# EPICS autosave request: xx_auto_scalcout_settings.req
$(P)$(S).A
$(P)$(S).B
$(P)$(S).C
$(P)$(S).D
$(P)$(S).E
$(P)$(S).F
$(P)$(S).G
$(P)$(S).H
$(P)$(S).I
$(P)$(S).J
$(P)$(S).K
$(P)$(S).L
$(P)$(S).INPA
$(P)$(S).INPB
$(P)$(S).INPC
$(P)$(S).INPD
$(P)$(S).INPE
$(P)$(S).INPF
$(P)$(S).INPG
$(P)$(S).INPH
$(P)$(S).INPI
$(P)$(S).INPJ
$(P)$(S).INPK
$(P)$(S).INPL
$(P)$(S).AA
$(P)$(S).BB
$(P)$(S).CC
$(P)$(S).DD
$(P)$(S).EE
$(P)$(S).FF
$(P)$(S).GG
$(P)$(S).HH
$(P)$(S).II
$(P)$(S).JJ
$(P)$(S).KK
$(P)$(S).LL
$(P)$(S).INAA
$(P)$(S).INBB
$(P)$(S).INCC
$(P)$(S).INDD
$(P)$(S).INEE
$(P)$(S).INFF
$(P)$(S).INGG
$(P)$(S).INHH
$(P)$(S).INII
$(P)$(S).INJJ
$(P)$(S).INKK
$(P)$(S).INLL
$(P)$(S).CALC
$(P)$(S).OCAL
$(P)$(S).SCAN
$(P)$(S).PREC
$(P)$(S).ODLY
$(P)$(S).OEVT
$(P)$(S).OOPT
$(P)$(S).DOPT
$(P)$(S).IVOA
$(P)$(S).IVOV
$(P)$(S).OUT
$(P)$(S).FLNK
$(P)$(S).DESC
$(P)$(S).EVNT
